{attribute 'qualified_only'}
{attribute 'strict'}
TYPE Action_list :
(
	idle := 0,
	clear_fault := 1,
	enable_all := 2,
	disable_all :=3,
	read_ncyl :=4,
	read_alias :=5,
	read_gains := 6,
	write_gains := 7,
	read_dongle_singlevalue := 8,
	save_soc_all := 9,
	bump_test := 10,
	function_generator := 11
) := idle;
END_TYPE

(* stored: Version 1.1.0.1, ProductVersion 3.1.4024.9
   EnumerationTextList Action_list: Id {b70eba98-7ca3-4256-9723-301bbc447da9} *)
